// TIA Portal V18 export
FUNCTION "recipe" : Void   // FC19, LAD
{ S7_Optimized_Access := 'TRUE' }
VERSION : 0.1
// stored: AutoNumber true, IsIECCheckEnabled false, SetENOAutomatically false, UDAEnableTagReadback false
BEGIN

REGION Network 1: program No from site
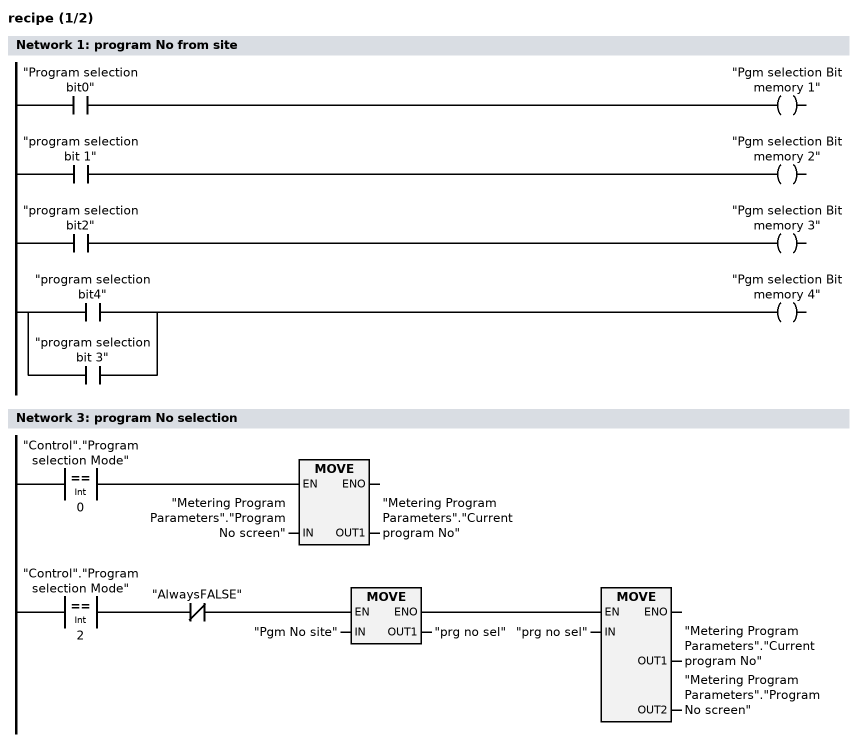
   RUNG wire#powerrail
      Contact( "Program selection bit0" )
      Coil( "Pgm selection Bit memory 1" )
   END_RUNG
   RUNG wire#powerrail
      Contact( "program selection bit 1" )
      Coil( "Pgm selection Bit memory 2" )
   END_RUNG
   RUNG wire#powerrail
      Contact( "program selection bit2" )
      Coil( "Pgm selection Bit memory 3" )
   END_RUNG
   RUNG wire#powerrail
      Contact( "program selection bit4" )
      wire#w1
      Coil( "Pgm selection Bit memory 4" )
   END_RUNG
   RUNG wire#powerrail
      Contact( "program selection bit 3" )
   END_RUNG wire#w1
   // the same network as SCL:
   "Pgm selection Bit memory 1" := "Program selection bit0";
   "Pgm selection Bit memory 2" := "program selection bit 1";
   "Pgm selection Bit memory 3" := "program selection bit2";
   "Pgm selection Bit memory 4" := "program selection bit4" OR "program selection bit 3";
END_REGION

REGION Network 2 (SCL)
   IF "Control"."Program selection Mode" = 1 THEN
     IF "Pgm selection Bit memory 1" THEN
       "Metering Program Parameters"."Receipe Program No" := 1;
     ELSIF "Pgm selection Bit memory 2" THEN
       "Metering Program Parameters"."Receipe Program No" := 2;
     ELSIF "Pgm selection Bit memory 3" THEN
       "Metering Program Parameters"."Receipe Program No" := 3;
     ELSIF "Pgm selection Bit memory 4" THEN
       "Metering Program Parameters"."Receipe Program No" := 4;
     ELSE
       "Metering Program Parameters"."Receipe Program No" := 0;
     END_IF;
   END_IF;
END_REGION

REGION Network 3: program No selection
   RUNG wire#powerrail
      { S7_Templates := "SrcType := Int" } EQ_Contact(in1 := "Control"."Program selection Mode", in2 := 0)
      Move(in := "Metering Program Parameters"."Program No screen", out1 => "Metering Program Parameters"."Current program No")
   END_RUNG
   RUNG wire#powerrail
      { S7_Templates := "SrcType := Int" } EQ_Contact(in1 := "Control"."Program selection Mode", in2 := 2)
      I_Contact( "AlwaysFALSE" )
      Move(in := "Pgm No site", out1 => "prg no sel")
      Move(in := "prg no sel", out1 => "Metering Program Parameters"."Current program No", out2 => "Metering Program Parameters"."Program No screen")
   END_RUNG
   // the same network as SCL:
   IF "Control"."Program selection Mode" = 0 THEN
       "Metering Program Parameters"."Current program No" := "Metering Program Parameters"."Program No screen";
   END_IF;
   IF ("Control"."Program selection Mode" = 2) AND NOT "AlwaysFALSE" THEN
       "prg no sel" := "Pgm No site";
       "Metering Program Parameters"."Current program No" := "prg no sel";
       "Metering Program Parameters"."Program No screen" := "prg no sel";
   END_IF;
END_REGION

REGION Network 4: Current flowrate qty and flowrate adjustment
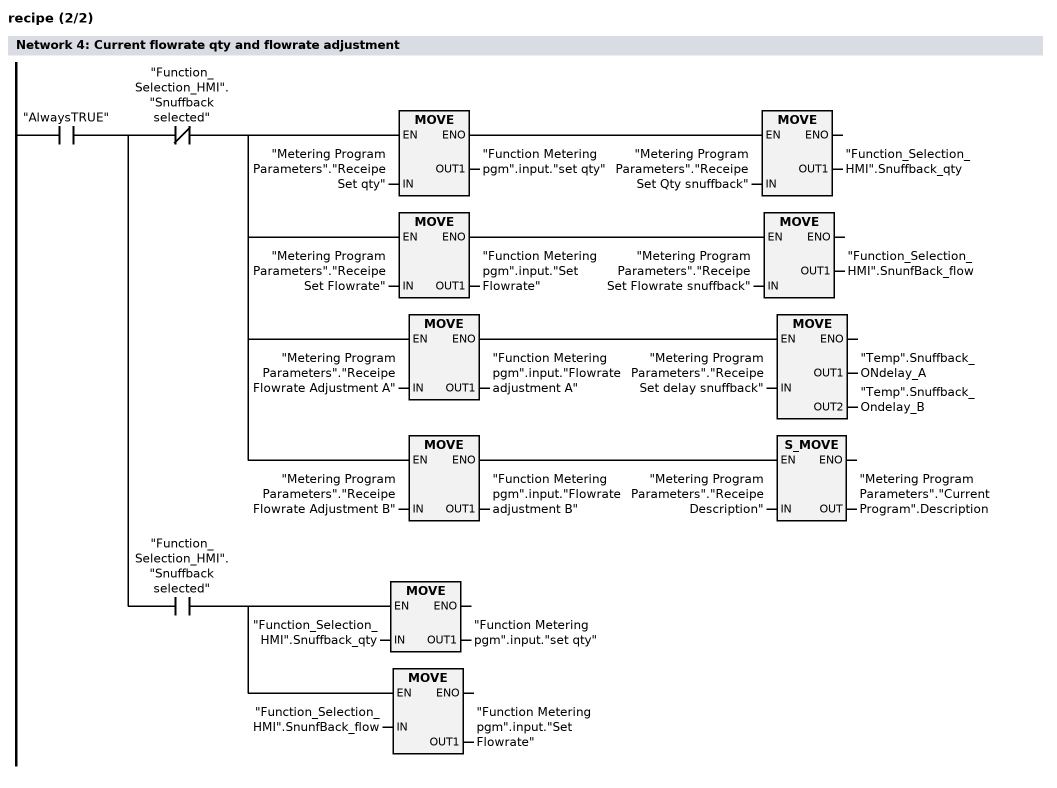
   RUNG wire#powerrail
      Contact( "AlwaysTRUE" )
      wire#w1
      I_Contact( "Function_Selection_HMI"."Snuffback selected" )
      wire#w2
      Move(in := "Metering Program Parameters"."Receipe Set qty", out1 => "Function Metering pgm".input."set qty")
      Move(in := "Metering Program Parameters"."Receipe Set Qty snuffback", out1 => "Function_Selection_HMI".Snuffback_qty)
   END_RUNG
   RUNG wire#w2
      Move(in := "Metering Program Parameters"."Receipe Set Flowrate", out1 => "Function Metering pgm".input."Set Flowrate")
      Move(in := "Metering Program Parameters"."Receipe Set Flowrate snuffback", out1 => "Function_Selection_HMI".SnunfBack_flow)
   END_RUNG
   RUNG wire#w2
      Move(in := "Metering Program Parameters"."Receipe Flowrate Adjustment A", out1 => "Function Metering pgm".input."Flowrate adjustment A")
      Move(in := "Metering Program Parameters"."Receipe Set delay snuffback", out1 => "Temp".Snuffback_ONdelay_A, out2 => "Temp".Snuffback_Ondelay_B)
   END_RUNG
   RUNG wire#w2
      Move(in := "Metering Program Parameters"."Receipe Flowrate Adjustment B", out1 => "Function Metering pgm".input."Flowrate adjustment B")
      S_Move(in := "Metering Program Parameters"."Receipe Description", out => "Metering Program Parameters"."Current Program".Description)
   END_RUNG
   RUNG wire#w1
      Contact( "Function_Selection_HMI"."Snuffback selected" )
      wire#w3
      Move(in := "Function_Selection_HMI".Snuffback_qty, out1 => "Function Metering pgm".input."set qty")
   END_RUNG
   RUNG wire#w3
      Move(in := "Function_Selection_HMI".SnunfBack_flow, out1 => "Function Metering pgm".input."Set Flowrate")
   END_RUNG
   // the same network as SCL:
   IF "AlwaysTRUE" AND NOT "Function_Selection_HMI"."Snuffback selected" THEN
       "Function Metering pgm".input."set qty" := "Metering Program Parameters"."Receipe Set qty";
       "Function_Selection_HMI".Snuffback_qty := "Metering Program Parameters"."Receipe Set Qty snuffback";
       "Function Metering pgm".input."Set Flowrate" := "Metering Program Parameters"."Receipe Set Flowrate";
       "Function_Selection_HMI".SnunfBack_flow := "Metering Program Parameters"."Receipe Set Flowrate snuffback";
       "Function Metering pgm".input."Flowrate adjustment A" := "Metering Program Parameters"."Receipe Flowrate Adjustment A";
       "Temp".Snuffback_ONdelay_A := "Metering Program Parameters"."Receipe Set delay snuffback";
       "Temp".Snuffback_Ondelay_B := "Metering Program Parameters"."Receipe Set delay snuffback";
       "Function Metering pgm".input."Flowrate adjustment B" := "Metering Program Parameters"."Receipe Flowrate Adjustment B";
       "Metering Program Parameters"."Current Program".Description := "Metering Program Parameters"."Receipe Description";
   END_IF;
   IF "AlwaysTRUE" AND "Function_Selection_HMI"."Snuffback selected" THEN
       "Function Metering pgm".input."set qty" := "Function_Selection_HMI".Snuffback_qty;
       "Function Metering pgm".input."Set Flowrate" := "Function_Selection_HMI".SnunfBack_flow;
   END_IF;
END_REGION
END_FUNCTION
